FUNCTION ScaledValue : REAL
VAR_INPUT
	mv : MonitoredValue;
END_VAR
VAR
END_VAR

IF (mv.rawValueMax - mv.rawValueMin) > 0 THEN
	ScaledValue := mv.scaledValueMin + (mv.rawValue - mv.rawValueMin) * ((mv.scaledValueMax- mv.scaledValueMin) / (mv.rawValueMax - mv.rawValueMin));
END_IF

END_FUNCTION

(* stored: Version 1.1.0.1, ProductVersion 3.1.4024.12
   POU ScaledValue: Id {e448d998-e884-4556-8621-1cf4500fd7e7}, SpecialFunc None *)
